FUNCTION_BLOCK FB_Elevation
VAR_INPUT
END_VAR
VAR_OUTPUT
END_VAR
VAR
	
	//Data for ADS communtication
	Targetpos_mm 			: LREAL	:= 0;		//Data FROM ADS
	Current_Position_mm 	: LREAL;			//Data TO ADS
	Enable AT %Q* 			: BOOL 	:= FALSE;	//Data FROM ADS
	Homeing 				: BOOL 	:= FALSE;	//Data TO ADS
	Homeing_Error 			: BOOL 	:= FALSE;	//Data TO ADS
	Homeing_Wrong_direction : BOOL  := FALSE;	//Data TO ADS
	Reset_requested 		: BOOL  := FALSE;	//Data FROM ADS
	Error AT %I* 			: BOOL;				//Data TO ADS
	//Position_Error AT %I* 	: BOOL;
	
	//Data for ADS communtication END
	
	
	Reset AT %Q* 			: BOOL 	:= FALSE;
	Encoder_Value AT %I* : UDINT;
	Homing_Switch AT %I* : BOOL;
	Limit_Switch AT %I* : BOOL;
	Warning AT %I* : BOOL;

	Ready AT %I* : BOOL;
	Moving_positive AT %I* : BOOL;
	Moving_negative AT %I* : BOOL;
	//In_target AT %I* : BOOL;
	Set_Encoder AT %Q* : BOOL;
	Encoder_Setvalue AT %Q* : UDINT;
	Target_Position AT %Q* : UDINT;
	
	//firstrun :BOOL := TRUE;
	Homed : BOOL := FALSE;
	Homeing_Allowed : BOOL := TRUE;
	Homeing_State : UINT := 0;
	Reset_state : UINT := 0;
	
	Homing_started_mm : LREAL; // to monitor if the homeing goes the right direction
	
	Homeing_Timer : TON; //used for timeouts
	Homeing_Timer2 : TON;
END_VAR

VAR CONSTANT
	maxmove_mm : LREAL := 210;
	minmove_mm : LREAL := 0;
	Zeroposition : UDINT := 1000000;
END_VAR

IF Homeing_Error THEN
	enable := FALSE;
	Homeing_state := 0;
	Homed := FALSE;
END_IF

IF Reset_requested THEN
	Reset_Elevation();
END_IF

IF Homed = FALSE AND Enable = TRUE AND Homeing_Allowed AND Homeing_Error = FALSE THEN
	//The homing sequence should start automaticly if the PLC is restarted and Enable is set
	Homeing_sequence();
ELSE
	IF Homed = TRUE AND Enable = TRUE THEN //Normal operation
		Target_Position := mm_to_encoder(LIMIT(minmove_mm,targetpos_mm,maxmove_mm));
	END_IF
END_IF

current_position_mm := encoder_to_mm(Encoder_Value);

METHOD encoder_to_mm : LREAL
VAR_INPUT
	encoder_pos : UDINT;
END_VAR

VAR
	encoder_ppr : LREAL := 2000;
	mm_per_rev : LREAL := 0.8; //calibrate this value
END_VAR
encoder_to_mm := UDINT_TO_LREAL(encoder_pos - Zeroposition) / (encoder_ppr * mm_per_rev);
END_METHOD

METHOD Homeing_sequence : BOOL
VAR_INPUT
END_VAR
VAR
	diff_pos : LREAL;
END_VAR
Homeing_Timer(IN:=TRUE, PT:= T#200S); //timeout of the homeing, it takes a long time to home...
Homeing := TRUE;

IF Homeing_Timer.Q THEN
	//Timeout as been reached
	Homeing_Error := TRUE;
	Homeing_Timer(IN:=FALSE);

END_IF

IF Homing_Switch AND Homeing_state < 3 THEN
	Homeing_state := 3;
END_IF

CASE Homeing_state OF
	0:
	 	//We want to set the current position to a high number so we can go into the negative as the countervalue is a UDINT
		Encoder_Setvalue := Zeroposition;
		Target_Position  := Zeroposition;
		Set_Encoder := 1;
		Homeing_Timer2(IN:= TRUE, PT:= T#1S);
		IF Homeing_Timer2.Q THEN
			Homeing_Timer2(IN:=FALSE);
			Homeing_state := 1;
		END_IF
			
	1:
		Set_Encoder := 0;
		
		Homeing_Timer2(IN:= TRUE, PT:= T#1S);
		IF Homeing_Timer2.Q THEN
			Homeing_Timer2(IN:=FALSE);
			Homeing_state := 2;
			Homing_started_mm := encoder_to_mm(Encoder_Value);
		END_IF
	2: 
		//Goes to a position in the 'negatives' 
		Target_Position := 0;
		diff_pos := (encoder_to_mm(Encoder_Value) - Homing_started_mm);
		//Diff_pos will be very large if it is going the correct direction due to underflow
		//If it does not grow large, it is going the wrong way 
		IF  diff_pos > 1 AND diff_pos < 1000 THEN
			// for some reason this happens sometime
			homeing_error := TRUE;
			Homeing_Wrong_direction := TRUE;
		END_IF
		
	3: 
		//Stop the motor and set the new zero when the motor has stopped
		Target_Position := Encoder_Value; //Stop the motor without disabling it
		Homeing_Timer2(IN:= TRUE, PT:= T#2S);
		IF Homeing_Timer2.Q THEN
			Encoder_Setvalue := Zeroposition;
			Target_Position := Zeroposition;
			Set_Encoder := 1;
			Homeing_state := 4;
			Homeing_Timer2(IN:=FALSE);
		END_IF
		
	4: 
	
		//Motor has been homed
		Set_Encoder := 0;
		Homeing_Timer(IN:=FALSE);
		Homeing := FALSE;
		Homed := TRUE;
		homeing_state := 0;
		
	
END_CASE
END_METHOD

METHOD mm_to_encoder : UDINT
VAR_INPUT
	mm_in : LREAL;
END_VAR
VAR
	encoder_ppr : LREAL := 2000;
	mm_per_rev : LREAL := 0.8; //calibrate this value
END_VAR
mm_to_encoder := LREAL_TO_UDINT(mm_in* mm_per_rev * encoder_ppr) + Zeroposition;
END_METHOD

METHOD Reset_Elevation : BOOL
VAR_INPUT
END_VAR

CASE Reset_state OF
	0:
		enable := FALSE;
		Reset_state := 1;
	1:
		Reset := TRUE;
		Targetpos_mm := Current_Position_mm ;
		Homed := FALSE;
		Homeing_Error := FALSE;
		Homeing_Wrong_direction := FALSE;
		Homeing_State := 0;
		Reset_state := 2;
		
	2: 
		Reset := FALSE;
		Reset_state := 3;
		
	3: //A extra one for good luck
		Reset := TRUE;
		Reset_state := 3;
		
	4: 
		Reset := FALSE;
		Reset_state := 0;
		Reset_requested := FALSE;
	
END_CASE
END_METHOD

END_FUNCTION_BLOCK

(* stored: Version 1.1.0.1, ProductVersion 3.1.4024.15
   POU FB_Elevation: Id {1bcf21b4-a4db-40ba-b81d-4360d1896368}, SpecialFunc None
   Method encoder_to_mm: Id {b5c4ff8f-17fb-45ab-a21d-86864561b433}
   Method Homeing_sequence: Id {0dc89b1f-92b0-4e40-988b-ba0866669870}
   Method mm_to_encoder: Id {595ffc56-8fd9-4170-a03c-9394cd1a5d9b}
   Method Reset_Elevation: Id {464d2e81-fada-4de1-a023-e78299ddcd83} *)
